{attribute 'qualified_only'}
{attribute 'strict'}
{attribute 'to_string'}
TYPE E_EtherCATMaster :
(
	Device2_EtherCAT		:=2,
	Device6_EtherCAT		:=6
);
END_TYPE

(* stored: Version 1.1.0.1, ProductVersion 3.1.4026.18
   DUT E_EtherCATMaster: Id {dc676ea9-0cca-4807-acc9-60b60199f493} *)
